// SIMATIC S7-200 project (STEP 7-Micro/WIN), CPU 221 REL 01.10

ORGANIZATION_BLOCK MAIN:OB1
TITLE=PROGRAM COMMENTS
BEGIN
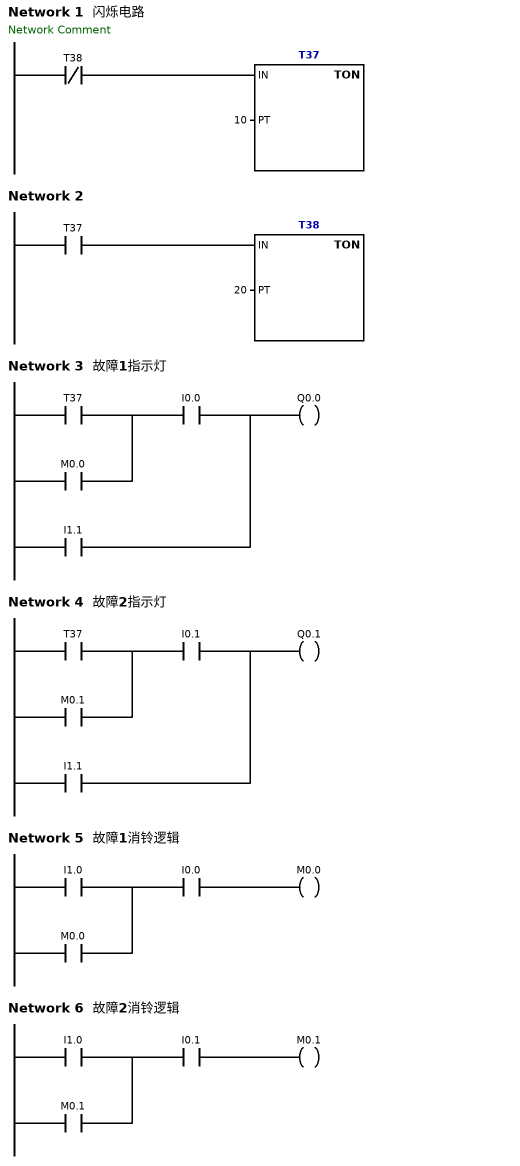
Network 1 // 闪烁电路
// Network Comment
// (network saved uncompiled; LAD cells follow)
// row 0: c0 -|/|- T38  c1 --  c2 [TON T37 IN:=power@row0, PT:=10]
// row 1: c2 [box]
Network 2
// (network saved uncompiled; LAD cells follow)
// row 0: c0 -| |- T37  c1 --  c2 [TON T38 IN:=power@row0, PT:=20]
// row 1: c2 [box]
Network 3 // 故障1指示灯
// (network saved uncompiled; LAD cells follow)
// row 0: c0 -| |- T37 v  c1 -| |- I0.0 v  c2 -( ) Q0.0
// row 1: c0 -| |- M0.0 ^  c1 ^v
// row 2: c0 -| |- I1.1  c1 -- ^
Network 4 // 故障2指示灯
// (network saved uncompiled; LAD cells follow)
// row 0: c0 -| |- T37 v  c1 -| |- I0.1 v  c2 -( ) Q0.1
// row 1: c0 -| |- M0.1 ^  c1 ^v
// row 2: c0 -| |- I1.1  c1 -- ^
Network 5 // 故障1消铃逻辑
// (network saved uncompiled; LAD cells follow)
// row 0: c0 -| |- I1.0 v  c1 -| |- I0.0  c2 -( ) M0.0
// row 1: c0 -| |- M0.0 ^
Network 6 // 故障2消铃逻辑
// (network saved uncompiled; LAD cells follow)
// row 0: c0 -| |- I1.0 v  c1 -| |- I0.1  c2 -( ) M0.1
// row 1: c0 -| |- M0.1 ^
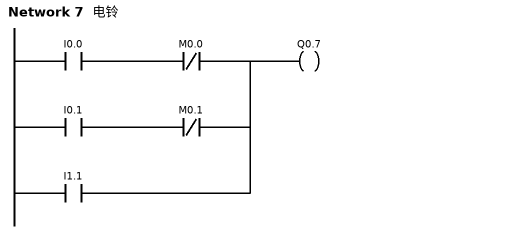
Network 7 // 电铃
// (network saved uncompiled; LAD cells follow)
// row 0: c0 -| |- I0.0  c1 -|/|- M0.0 v  c2 -( ) Q0.7
// row 1: c0 -| |- I0.1  c1 -|/|- M0.1 ^v
// row 2: c0 -| |- I1.1  c1 -- ^
END_ORGANIZATION_BLOCK
